TYPE ST_AuditLogMessages :
    STRUCT
        Timestamp : T_MaxString;
        k   : T_MaxString;
        v   : T_MaxString;	
    END_STRUCT
END_TYPE

(* stored: Version 1.1.0.1
   DUT ST_AuditLogMessages: Id {4ca4baac-e387-4596-b590-35a258f2dcc3} *)
